// TIA Portal V20 export
TYPE "LConSMC_typeLoadGear"
// stored: Access Published
   STRUCT
      numerator : UDInt := 1;   // Anzahl an Motorumdrehungen / Number of motor revolutions
      denominator : UDInt := 1;   // Anzahl an Lastumdrehungen / Number of load revolutions
   END_STRUCT;
END_TYPE
